FUNCTION_BLOCK FB_SequenceControl (* Basic Function Block Type *)
  (* Standard: 61499-2 *)
  (* Version 0.0, 2014-5-4, wildai, nxtControl GmbH, Template *)
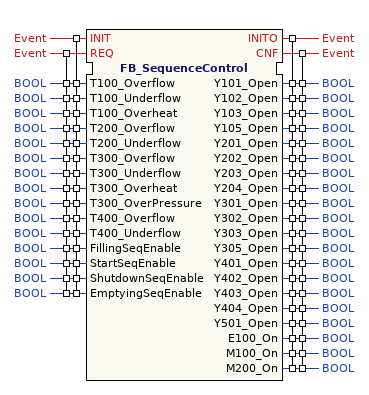
  EVENT_INPUT
    INIT WITH T100_Overflow, T100_Underflow, T100_Overheat, T200_Overflow, T200_Underflow, T300_Overflow, T300_Underflow, T300_Overheat, T300_OverPressure, T400_Overflow, T400_Underflow, FillingSeqEnable, StartSeqEnable, ShutdownSeqEnable, EmptyingSeqEnable; (* Initialization Request *)
    REQ WITH T100_Overflow, T100_Underflow, T100_Overheat, T200_Overflow, T200_Underflow, T300_Overflow, T300_Underflow, T300_Overheat, T300_OverPressure, T400_Overflow, T400_Underflow, FillingSeqEnable, StartSeqEnable, ShutdownSeqEnable, EmptyingSeqEnable; (* Normal Execution Request *)
  END_EVENT
  EVENT_OUTPUT
    INITO WITH Y101_Open, Y102_Open, Y103_Open, Y105_Open, Y201_Open, Y202_Open, Y203_Open, Y204_Open, Y301_Open, Y302_Open, Y303_Open, Y305_Open, Y401_Open, Y402_Open, Y403_Open, Y404_Open, Y501_Open, E100_On, M100_On, M200_On; (* Initialization Confirm *)
    CNF WITH Y101_Open, Y102_Open, Y103_Open, Y105_Open, Y201_Open, Y202_Open, Y203_Open, Y204_Open, Y301_Open, Y302_Open, Y303_Open, Y305_Open, Y401_Open, Y402_Open, Y403_Open, Y404_Open, Y501_Open, E100_On, M100_On, M200_On; (* Execution Confirmation *)
  END_EVENT
  VAR_INPUT
    T100_Overflow : BOOL;
    T100_Underflow : BOOL;
    T100_Overheat : BOOL;
    T200_Overflow : BOOL;
    T200_Underflow : BOOL;
    T300_Overflow : BOOL;
    T300_Underflow : BOOL;
    T300_Overheat : BOOL;
    T300_OverPressure : BOOL;
    T400_Overflow : BOOL;
    T400_Underflow : BOOL;
    FillingSeqEnable : BOOL;
    StartSeqEnable : BOOL;
    ShutdownSeqEnable : BOOL;
    EmptyingSeqEnable : BOOL;
  END_VAR
  VAR_OUTPUT
    Y101_Open : BOOL;
    Y102_Open : BOOL;
    Y103_Open : BOOL;
    Y105_Open : BOOL;
    Y201_Open : BOOL;
    Y202_Open : BOOL;
    Y203_Open : BOOL;
    Y204_Open : BOOL;
    Y301_Open : BOOL;
    Y302_Open : BOOL;
    Y303_Open : BOOL;
    Y305_Open : BOOL;
    Y401_Open : BOOL;
    Y402_Open : BOOL;
    Y403_Open : BOOL;
    Y404_Open : BOOL;
    Y501_Open : BOOL;
    E100_On : BOOL;
    M100_On : BOOL;
    M200_On : BOOL;
  END_VAR
  VAR
    FillingSeqComplete : BOOL;
    StartSeqComplete : BOOL;
    EmptyingComplete : BOOL;
  END_VAR
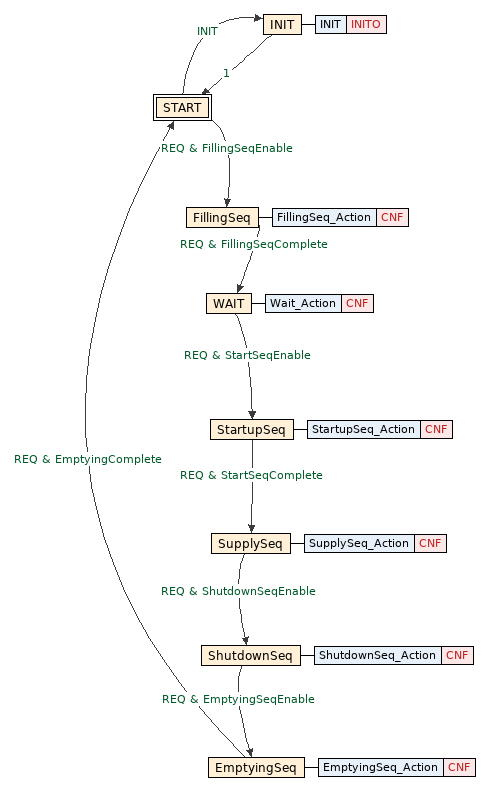
  EC_STATES
    START; (* Initial State *)
    INIT : INIT -> INITO; (* Initialization *)
    FillingSeq : FillingSeq_Action -> CNF; (* Normal execution *)
    WAIT : Wait_Action -> CNF;
    StartupSeq : StartupSeq_Action -> CNF;
    SupplySeq : SupplySeq_Action -> CNF;
    ShutdownSeq : ShutdownSeq_Action -> CNF;
    EmptyingSeq : EmptyingSeq_Action -> CNF;
  END_STATES
  EC_TRANSITIONS
    START TO INIT := INIT;
    INIT TO START := 1;
    START TO FillingSeq := REQ & FillingSeqEnable;
    FillingSeq TO WAIT := REQ & FillingSeqComplete;
    WAIT TO StartupSeq := REQ & StartSeqEnable;
    StartupSeq TO SupplySeq := REQ & StartSeqComplete;
    SupplySeq TO ShutdownSeq := REQ & ShutdownSeqEnable;
    ShutdownSeq TO EmptyingSeq := REQ & EmptyingSeqEnable;
    EmptyingSeq TO START := REQ & EmptyingComplete;
  END_TRANSITIONS
  ALGORITHM INIT IN ST: (* Initialization algorithm *)
;

Y101_Open := FALSE;
Y102_Open := FALSE;
Y103_Open := FALSE;
Y105_Open := FALSE;
Y201_Open := FALSE;
Y202_Open := FALSE;
Y203_Open := FALSE;
Y204_Open := TRUE; /*For Over Pressure */
Y301_Open := FALSE;
Y302_Open := FALSE;
Y303_Open := FALSE;
Y305_Open := FALSE;
Y401_Open := FALSE;
Y402_Open := FALSE;
Y403_Open := FALSE;
Y404_Open := FALSE;
Y501_Open := FALSE;
E100_On := FALSE;
M100_On := FALSE;
M200_On := FALSE;
  END_ALGORITHM
  ALGORITHM FillingSeq_Action IN ST:
;

Y101_Open := TRUE;
Y102_Open := TRUE;
M100_On := TRUE;
Y203_Open := TRUE;
Y201_Open := TRUE;
M200_On := TRUE;
Y303_Open := TRUE;
Y301_Open := TRUE;

FillingSeqComplete := NOT (T100_Underflow OR T200_Underflow OR T300_Underflow OR T400_Underflow);
  END_ALGORITHM
  ALGORITHM EmptyingSeq_Action IN ST:
;

IF NOT T400_Underflow THEN
	Y105_Open := TRUE;
END_IF;

IF NOT T200_Underflow THEN
	Y201_Open := TRUE;
	M200_On := TRUE;
	Y303_Open := TRUE;
	Y301_Open := TRUE;
END_IF;

IF NOT T300_Underflow THEN
	Y305_Open := TRUE;
	Y501_Open := TRUE;
END_IF

IF NOT T400_Underflow THEN
	Y101_Open := TRUE;
END_IF;

EmptyingComplete := T100_Underflow AND T200_Underflow AND T300_Underflow AND T400_Underflow;
  END_ALGORITHM
  ALGORITHM ShutdownSeq_Action IN ST:
;

Y501_Open := FALSE;
E100_On := FALSE;
Y102_Open := FALSE;
M100_On := FALSE;
Y203_Open := FALSE;
Y201_Open := FALSE;
M200_On := FALSE;
Y303_Open := FALSE;
Y301_Open := FALSE;
Y305_Open := FALSE;
  END_ALGORITHM
  ALGORITHM StartupSeq_Action IN ST:
;

Y101_Open := FALSE;
Y102_Open := FALSE;
Y103_Open := FALSE;
Y105_Open := FALSE;
Y201_Open := FALSE;
Y202_Open := FALSE;
Y203_Open := FALSE;
Y204_Open := TRUE;  /* For Over Pressure */
Y301_Open := FALSE;
Y302_Open := FALSE;
Y303_Open := FALSE;
Y305_Open := FALSE;
Y401_Open := FALSE;
Y402_Open := FALSE;
Y403_Open := FALSE;
Y404_Open := FALSE;
Y501_Open := FALSE;
E100_On := FALSE;
M100_On := FALSE;
M200_On := FALSE;
  END_ALGORITHM
  ALGORITHM SupplySeq_Action IN ST:
;

Y501_Open := TRUE;
  END_ALGORITHM
  ALGORITHM Wait_Action IN ST:
;

Y101_Open := FALSE;
Y102_Open := FALSE;
M100_On := FALSE;
Y203_Open := FALSE;
Y201_Open := FALSE;
M200_On := FALSE;
Y303_Open := FALSE;
Y301_Open := FALSE;
  END_ALGORITHM
END_FUNCTION_BLOCK
